Fanuc TP program (LS listing): GRIPPER_CONTROL.ls

/PROG  GRIPPER_CONTROL
/ATTR
OWNER   = MNEDITOR;
COMMENT   = "OR Gripper Move";
PROG_SIZE = 1050;
CREATE    = DATE 18-01-21  TIME 12:00:00;
MODIFIED  = DATE 18-01-21  TIME 12:00:00;
FILE_NAME = ;
VERSION   = 0;
LINE_COUNT  = 30;
MEMORY_SIZE = 1310;
PROTECT   = READ_WRITE;
TCD:  STACK_SIZE  = 0,
      TASK_PRIORITY = 50,
      TIME_SLICE  = 0,
      BUSY_LAMP_OFF = 0,
      ABORT_REQUEST = 0,
      PAUSE_REQUEST = 0;
DEFAULT_GROUP = *,*,*,*,*;
CONTROL_CODE  = 00000000 00000000;
/MN
    :  !set wait flag to 0 as calling KAREL routine is not affected by  it anyways;
    :  CALL IPL_OR_RG_MOVE(R[81], R[82], 0);
/END
